% RSLogix 500 project semaforo.RSS, saved by version 8.40.00.08 %
PROJECT "UNTITLED"    % processor: MicroLogix 1500 %

PROGRAM FILES
  LAD 2   3 rungs

DATA FILES
  O0 OUTPUT  4 elements
  I1 INPUT  5 elements
  S2 STATUS  66 elements
  B3 BINARY  1 elements
  T4 TIMER  3 elements
  C5 COUNTER  1 elements
  R6 CONTROL  1 elements
  N7 INTEGER  1 elements
  F8 FLOAT  1 elements

LADDER 2
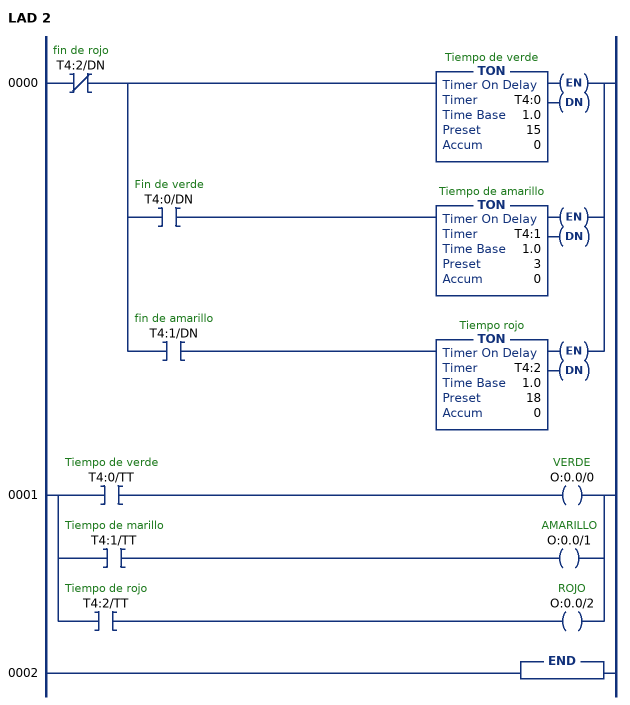
% Rung: 0 %
SOR XIO T4:2/DN BST TON T4:0 1.0 15 0 NXB XIC T4:0/DN TON T4:1 1.0 3 0 NXB XIC T4:1/DN TON T4:2 1.0 18 0 BND EOR
%   T4:2/DN  "fin de rojo" %
%   T4:0  "Tiempo de verde" %
%   T4:0/DN  "Fin de verde" %
%   T4:1  "Tiempo de amarillo" %
%   T4:1/DN  "fin de amarillo" %
%   T4:2  "Tiempo rojo" %
% Rung: 1 %
SOR BST XIC T4:0/TT OTE O:0.0/0 NXB XIC T4:1/TT OTE O:0.0/1 NXB XIC T4:2/TT OTE O:0.0/2 BND EOR
%   T4:0/TT  "Tiempo de verde" %
%   O:0.0/0  VERDE %
%   T4:1/TT  "Tiempo de marillo" %
%   O:0.0/1  AMARILLO %
%   T4:2/TT  "Tiempo de rojo" %
%   O:0.0/2  ROJO %
% Rung: 2 %
SOR END EOR

DATA TABLE (non-zero values as saved)
DATA T4
% .PRE .ACC %
% T4:0 % 15 0
% T4:1 % 3 0
% T4:2 % 18 0
